(* IEC 61131-3 sources: TA/Tests/RetainTest/At (part 6) *)

(* ---- AtRetainStructureSimple.st ---- *)
PROGRAM AtRetainStructureSimple

AT_RETAINTEST_RETAIN_STRUCTURESIMPLE.AUTO2_BOOL := AT_RETAINTEST_RETAIN_STRUCTURESIMPLE.AUTO1_BOOL;
AT_RETAINTEST_RETAIN_STRUCTURESIMPLE.AUTO2_BYTE := AT_RETAINTEST_RETAIN_STRUCTURESIMPLE.AUTO1_BYTE;
AT_RETAINTEST_RETAIN_STRUCTURESIMPLE.AUTO2_DATE := AT_RETAINTEST_RETAIN_STRUCTURESIMPLE.AUTO1_DATE;
AT_RETAINTEST_RETAIN_STRUCTURESIMPLE.AUTO2_DINT := AT_RETAINTEST_RETAIN_STRUCTURESIMPLE.AUTO1_DINT;
AT_RETAINTEST_RETAIN_STRUCTURESIMPLE.AUTO2_DWORD := AT_RETAINTEST_RETAIN_STRUCTURESIMPLE.AUTO1_DWORD;
AT_RETAINTEST_RETAIN_STRUCTURESIMPLE.AUTO2_INT := AT_RETAINTEST_RETAIN_STRUCTURESIMPLE.AUTO1_INT;
AT_RETAINTEST_RETAIN_STRUCTURESIMPLE.AUTO2_LINT := AT_RETAINTEST_RETAIN_STRUCTURESIMPLE.AUTO1_LINT;
AT_RETAINTEST_RETAIN_STRUCTURESIMPLE.AUTO2_LREAL := AT_RETAINTEST_RETAIN_STRUCTURESIMPLE.AUTO1_LREAL;
AT_RETAINTEST_RETAIN_STRUCTURESIMPLE.AUTO2_LWORD := AT_RETAINTEST_RETAIN_STRUCTURESIMPLE.AUTO1_LWORD;
AT_RETAINTEST_RETAIN_STRUCTURESIMPLE.AUTO2_REAL := AT_RETAINTEST_RETAIN_STRUCTURESIMPLE.AUTO1_REAL;
AT_RETAINTEST_RETAIN_STRUCTURESIMPLE.AUTO2_SINT := AT_RETAINTEST_RETAIN_STRUCTURESIMPLE.AUTO1_SINT;
AT_RETAINTEST_RETAIN_STRUCTURESIMPLE.AUTO2_STRING := AT_RETAINTEST_RETAIN_STRUCTURESIMPLE.AUTO1_STRING;
AT_RETAINTEST_RETAIN_STRUCTURESIMPLE.AUTO2_TIME := AT_RETAINTEST_RETAIN_STRUCTURESIMPLE.AUTO1_TIME;
AT_RETAINTEST_RETAIN_STRUCTURESIMPLE.AUTO2_UDINT := AT_RETAINTEST_RETAIN_STRUCTURESIMPLE.AUTO1_UDINT;
AT_RETAINTEST_RETAIN_STRUCTURESIMPLE.AUTO2_UINT := AT_RETAINTEST_RETAIN_STRUCTURESIMPLE.AUTO1_UINT;
AT_RETAINTEST_RETAIN_STRUCTURESIMPLE.AUTO2_ULINT := AT_RETAINTEST_RETAIN_STRUCTURESIMPLE.AUTO1_ULINT;
AT_RETAINTEST_RETAIN_STRUCTURESIMPLE.AUTO2_USINT := AT_RETAINTEST_RETAIN_STRUCTURESIMPLE.AUTO1_USINT;
AT_RETAINTEST_RETAIN_STRUCTURESIMPLE.AUTO2_WORD := AT_RETAINTEST_RETAIN_STRUCTURESIMPLE.AUTO1_WORD;

AT_RETAINTEST_NONRETAIN_STRUCTURESIMPLE.AUTO2_BOOL := AT_RETAINTEST_NONRETAIN_STRUCTURESIMPLE.AUTO1_BOOL;
AT_RETAINTEST_NONRETAIN_STRUCTURESIMPLE.AUTO2_BYTE := AT_RETAINTEST_NONRETAIN_STRUCTURESIMPLE.AUTO1_BYTE;
AT_RETAINTEST_NONRETAIN_STRUCTURESIMPLE.AUTO2_DATE := AT_RETAINTEST_NONRETAIN_STRUCTURESIMPLE.AUTO1_DATE;
AT_RETAINTEST_NONRETAIN_STRUCTURESIMPLE.AUTO2_DINT := AT_RETAINTEST_NONRETAIN_STRUCTURESIMPLE.AUTO1_DINT;
AT_RETAINTEST_NONRETAIN_STRUCTURESIMPLE.AUTO2_DWORD := AT_RETAINTEST_NONRETAIN_STRUCTURESIMPLE.AUTO1_DWORD;
AT_RETAINTEST_NONRETAIN_STRUCTURESIMPLE.AUTO2_INT := AT_RETAINTEST_NONRETAIN_STRUCTURESIMPLE.AUTO1_INT;
AT_RETAINTEST_NONRETAIN_STRUCTURESIMPLE.AUTO2_LINT := AT_RETAINTEST_NONRETAIN_STRUCTURESIMPLE.AUTO1_LINT;
AT_RETAINTEST_NONRETAIN_STRUCTURESIMPLE.AUTO2_LREAL := AT_RETAINTEST_NONRETAIN_STRUCTURESIMPLE.AUTO1_LREAL;
AT_RETAINTEST_NONRETAIN_STRUCTURESIMPLE.AUTO2_LWORD := AT_RETAINTEST_NONRETAIN_STRUCTURESIMPLE.AUTO1_LWORD;
AT_RETAINTEST_NONRETAIN_STRUCTURESIMPLE.AUTO2_REAL := AT_RETAINTEST_NONRETAIN_STRUCTURESIMPLE.AUTO1_REAL;
AT_RETAINTEST_NONRETAIN_STRUCTURESIMPLE.AUTO2_SINT := AT_RETAINTEST_NONRETAIN_STRUCTURESIMPLE.AUTO1_SINT;
AT_RETAINTEST_NONRETAIN_STRUCTURESIMPLE.AUTO2_STRING := AT_RETAINTEST_NONRETAIN_STRUCTURESIMPLE.AUTO1_STRING;
AT_RETAINTEST_NONRETAIN_STRUCTURESIMPLE.AUTO2_TIME := AT_RETAINTEST_NONRETAIN_STRUCTURESIMPLE.AUTO1_TIME;
AT_RETAINTEST_NONRETAIN_STRUCTURESIMPLE.AUTO2_UDINT := AT_RETAINTEST_NONRETAIN_STRUCTURESIMPLE.AUTO1_UDINT;
AT_RETAINTEST_NONRETAIN_STRUCTURESIMPLE.AUTO2_UINT := AT_RETAINTEST_NONRETAIN_STRUCTURESIMPLE.AUTO1_UINT;
AT_RETAINTEST_NONRETAIN_STRUCTURESIMPLE.AUTO2_ULINT := AT_RETAINTEST_NONRETAIN_STRUCTURESIMPLE.AUTO1_ULINT;
AT_RETAINTEST_NONRETAIN_STRUCTURESIMPLE.AUTO2_USINT := AT_RETAINTEST_NONRETAIN_STRUCTURESIMPLE.AUTO1_USINT;
AT_RETAINTEST_NONRETAIN_STRUCTURESIMPLE.AUTO2_WORD := AT_RETAINTEST_NONRETAIN_STRUCTURESIMPLE.AUTO1_WORD;

AT_RETAINTEST_AUTO_STRUCTURESIMPLE.AUTO2_BOOL := AT_RETAINTEST_AUTO_STRUCTURESIMPLE.AUTO1_BOOL;
AT_RETAINTEST_AUTO_STRUCTURESIMPLE.AUTO2_BYTE := AT_RETAINTEST_AUTO_STRUCTURESIMPLE.AUTO1_BYTE;
AT_RETAINTEST_AUTO_STRUCTURESIMPLE.AUTO2_DATE := AT_RETAINTEST_AUTO_STRUCTURESIMPLE.AUTO1_DATE;
AT_RETAINTEST_AUTO_STRUCTURESIMPLE.AUTO2_DINT := AT_RETAINTEST_AUTO_STRUCTURESIMPLE.AUTO1_DINT;
AT_RETAINTEST_AUTO_STRUCTURESIMPLE.AUTO2_DWORD := AT_RETAINTEST_AUTO_STRUCTURESIMPLE.AUTO1_DWORD;
AT_RETAINTEST_AUTO_STRUCTURESIMPLE.AUTO2_INT := AT_RETAINTEST_AUTO_STRUCTURESIMPLE.AUTO1_INT;
AT_RETAINTEST_AUTO_STRUCTURESIMPLE.AUTO2_LINT := AT_RETAINTEST_AUTO_STRUCTURESIMPLE.AUTO1_LINT;
AT_RETAINTEST_AUTO_STRUCTURESIMPLE.AUTO2_LREAL := AT_RETAINTEST_AUTO_STRUCTURESIMPLE.AUTO1_LREAL;
AT_RETAINTEST_AUTO_STRUCTURESIMPLE.AUTO2_LWORD := AT_RETAINTEST_AUTO_STRUCTURESIMPLE.AUTO1_LWORD;
AT_RETAINTEST_AUTO_STRUCTURESIMPLE.AUTO2_REAL := AT_RETAINTEST_AUTO_STRUCTURESIMPLE.AUTO1_REAL;
AT_RETAINTEST_AUTO_STRUCTURESIMPLE.AUTO2_SINT := AT_RETAINTEST_AUTO_STRUCTURESIMPLE.AUTO1_SINT;
AT_RETAINTEST_AUTO_STRUCTURESIMPLE.AUTO2_STRING := AT_RETAINTEST_AUTO_STRUCTURESIMPLE.AUTO1_STRING;
AT_RETAINTEST_AUTO_STRUCTURESIMPLE.AUTO2_TIME := AT_RETAINTEST_AUTO_STRUCTURESIMPLE.AUTO1_TIME;
AT_RETAINTEST_AUTO_STRUCTURESIMPLE.AUTO2_UDINT := AT_RETAINTEST_AUTO_STRUCTURESIMPLE.AUTO1_UDINT;
AT_RETAINTEST_AUTO_STRUCTURESIMPLE.AUTO2_UINT := AT_RETAINTEST_AUTO_STRUCTURESIMPLE.AUTO1_UINT;
AT_RETAINTEST_AUTO_STRUCTURESIMPLE.AUTO2_ULINT := AT_RETAINTEST_AUTO_STRUCTURESIMPLE.AUTO1_ULINT;
AT_RETAINTEST_AUTO_STRUCTURESIMPLE.AUTO2_USINT := AT_RETAINTEST_AUTO_STRUCTURESIMPLE.AUTO1_USINT;
AT_RETAINTEST_AUTO_STRUCTURESIMPLE.AUTO2_WORD := AT_RETAINTEST_AUTO_STRUCTURESIMPLE.AUTO1_WORD;

END_PROGRAM

(* ---- AtRetainStructureStructureSimple.st ---- *)
PROGRAM AtRetainStructureStructureSimple

AT_RETAINTEST_RETAIN_STRUCTURESTRUCTURESIMPLE.AUTO2.SIMPLE_BOOL := AT_RETAINTEST_RETAIN_STRUCTURESTRUCTURESIMPLE.AUTO1.SIMPLE_BOOL;
AT_RETAINTEST_RETAIN_STRUCTURESTRUCTURESIMPLE.AUTO2.SIMPLE_BYTE := AT_RETAINTEST_RETAIN_STRUCTURESTRUCTURESIMPLE.AUTO1.SIMPLE_BYTE;
AT_RETAINTEST_RETAIN_STRUCTURESTRUCTURESIMPLE.AUTO2.SIMPLE_DATE := AT_RETAINTEST_RETAIN_STRUCTURESTRUCTURESIMPLE.AUTO1.SIMPLE_DATE;
AT_RETAINTEST_RETAIN_STRUCTURESTRUCTURESIMPLE.AUTO2.SIMPLE_DINT := AT_RETAINTEST_RETAIN_STRUCTURESTRUCTURESIMPLE.AUTO1.SIMPLE_DINT;
AT_RETAINTEST_RETAIN_STRUCTURESTRUCTURESIMPLE.AUTO2.SIMPLE_DWORD := AT_RETAINTEST_RETAIN_STRUCTURESTRUCTURESIMPLE.AUTO1.SIMPLE_DWORD;
AT_RETAINTEST_RETAIN_STRUCTURESTRUCTURESIMPLE.AUTO2.SIMPLE_INT := AT_RETAINTEST_RETAIN_STRUCTURESTRUCTURESIMPLE.AUTO1.SIMPLE_INT;
AT_RETAINTEST_RETAIN_STRUCTURESTRUCTURESIMPLE.AUTO2.SIMPLE_LINT := AT_RETAINTEST_RETAIN_STRUCTURESTRUCTURESIMPLE.AUTO1.SIMPLE_LINT;
AT_RETAINTEST_RETAIN_STRUCTURESTRUCTURESIMPLE.AUTO2.SIMPLE_LREAL := AT_RETAINTEST_RETAIN_STRUCTURESTRUCTURESIMPLE.AUTO1.SIMPLE_LREAL;
AT_RETAINTEST_RETAIN_STRUCTURESTRUCTURESIMPLE.AUTO2.SIMPLE_LWORD := AT_RETAINTEST_RETAIN_STRUCTURESTRUCTURESIMPLE.AUTO1.SIMPLE_LWORD;
AT_RETAINTEST_RETAIN_STRUCTURESTRUCTURESIMPLE.AUTO2.SIMPLE_REAL := AT_RETAINTEST_RETAIN_STRUCTURESTRUCTURESIMPLE.AUTO1.SIMPLE_REAL;
AT_RETAINTEST_RETAIN_STRUCTURESTRUCTURESIMPLE.AUTO2.SIMPLE_SINT := AT_RETAINTEST_RETAIN_STRUCTURESTRUCTURESIMPLE.AUTO1.SIMPLE_SINT;
AT_RETAINTEST_RETAIN_STRUCTURESTRUCTURESIMPLE.AUTO2.SIMPLE_STRING := AT_RETAINTEST_RETAIN_STRUCTURESTRUCTURESIMPLE.AUTO1.SIMPLE_STRING;
AT_RETAINTEST_RETAIN_STRUCTURESTRUCTURESIMPLE.AUTO2.SIMPLE_TIME := AT_RETAINTEST_RETAIN_STRUCTURESTRUCTURESIMPLE.AUTO1.SIMPLE_TIME;
AT_RETAINTEST_RETAIN_STRUCTURESTRUCTURESIMPLE.AUTO2.SIMPLE_UDINT := AT_RETAINTEST_RETAIN_STRUCTURESTRUCTURESIMPLE.AUTO1.SIMPLE_UDINT;
AT_RETAINTEST_RETAIN_STRUCTURESTRUCTURESIMPLE.AUTO2.SIMPLE_UINT := AT_RETAINTEST_RETAIN_STRUCTURESTRUCTURESIMPLE.AUTO1.SIMPLE_UINT;
AT_RETAINTEST_RETAIN_STRUCTURESTRUCTURESIMPLE.AUTO2.SIMPLE_ULINT := AT_RETAINTEST_RETAIN_STRUCTURESTRUCTURESIMPLE.AUTO1.SIMPLE_ULINT;
AT_RETAINTEST_RETAIN_STRUCTURESTRUCTURESIMPLE.AUTO2.SIMPLE_USINT := AT_RETAINTEST_RETAIN_STRUCTURESTRUCTURESIMPLE.AUTO1.SIMPLE_USINT;
AT_RETAINTEST_RETAIN_STRUCTURESTRUCTURESIMPLE.AUTO2.SIMPLE_WORD := AT_RETAINTEST_RETAIN_STRUCTURESTRUCTURESIMPLE.AUTO1.SIMPLE_WORD;

AT_RETAINTEST_NONRETAIN_STRUCTURESTRUCTURESIMPLE.AUTO2.SIMPLE_BOOL := AT_RETAINTEST_NONRETAIN_STRUCTURESTRUCTURESIMPLE.AUTO1.SIMPLE_BOOL;
AT_RETAINTEST_NONRETAIN_STRUCTURESTRUCTURESIMPLE.AUTO2.SIMPLE_BYTE := AT_RETAINTEST_NONRETAIN_STRUCTURESTRUCTURESIMPLE.AUTO1.SIMPLE_BYTE;
AT_RETAINTEST_NONRETAIN_STRUCTURESTRUCTURESIMPLE.AUTO2.SIMPLE_DATE := AT_RETAINTEST_NONRETAIN_STRUCTURESTRUCTURESIMPLE.AUTO1.SIMPLE_DATE;
AT_RETAINTEST_NONRETAIN_STRUCTURESTRUCTURESIMPLE.AUTO2.SIMPLE_DINT := AT_RETAINTEST_NONRETAIN_STRUCTURESTRUCTURESIMPLE.AUTO1.SIMPLE_DINT;
AT_RETAINTEST_NONRETAIN_STRUCTURESTRUCTURESIMPLE.AUTO2.SIMPLE_DWORD := AT_RETAINTEST_NONRETAIN_STRUCTURESTRUCTURESIMPLE.AUTO1.SIMPLE_DWORD;
AT_RETAINTEST_NONRETAIN_STRUCTURESTRUCTURESIMPLE.AUTO2.SIMPLE_INT := AT_RETAINTEST_NONRETAIN_STRUCTURESTRUCTURESIMPLE.AUTO1.SIMPLE_INT;
AT_RETAINTEST_NONRETAIN_STRUCTURESTRUCTURESIMPLE.AUTO2.SIMPLE_LINT := AT_RETAINTEST_NONRETAIN_STRUCTURESTRUCTURESIMPLE.AUTO1.SIMPLE_LINT;
AT_RETAINTEST_NONRETAIN_STRUCTURESTRUCTURESIMPLE.AUTO2.SIMPLE_LREAL := AT_RETAINTEST_NONRETAIN_STRUCTURESTRUCTURESIMPLE.AUTO1.SIMPLE_LREAL;
AT_RETAINTEST_NONRETAIN_STRUCTURESTRUCTURESIMPLE.AUTO2.SIMPLE_LWORD := AT_RETAINTEST_NONRETAIN_STRUCTURESTRUCTURESIMPLE.AUTO1.SIMPLE_LWORD;
AT_RETAINTEST_NONRETAIN_STRUCTURESTRUCTURESIMPLE.AUTO2.SIMPLE_REAL := AT_RETAINTEST_NONRETAIN_STRUCTURESTRUCTURESIMPLE.AUTO1.SIMPLE_REAL;
AT_RETAINTEST_NONRETAIN_STRUCTURESTRUCTURESIMPLE.AUTO2.SIMPLE_SINT := AT_RETAINTEST_NONRETAIN_STRUCTURESTRUCTURESIMPLE.AUTO1.SIMPLE_SINT;
AT_RETAINTEST_NONRETAIN_STRUCTURESTRUCTURESIMPLE.AUTO2.SIMPLE_STRING := AT_RETAINTEST_NONRETAIN_STRUCTURESTRUCTURESIMPLE.AUTO1.SIMPLE_STRING;
AT_RETAINTEST_NONRETAIN_STRUCTURESTRUCTURESIMPLE.AUTO2.SIMPLE_TIME := AT_RETAINTEST_NONRETAIN_STRUCTURESTRUCTURESIMPLE.AUTO1.SIMPLE_TIME;
AT_RETAINTEST_NONRETAIN_STRUCTURESTRUCTURESIMPLE.AUTO2.SIMPLE_UDINT := AT_RETAINTEST_NONRETAIN_STRUCTURESTRUCTURESIMPLE.AUTO1.SIMPLE_UDINT;
AT_RETAINTEST_NONRETAIN_STRUCTURESTRUCTURESIMPLE.AUTO2.SIMPLE_UINT := AT_RETAINTEST_NONRETAIN_STRUCTURESTRUCTURESIMPLE.AUTO1.SIMPLE_UINT;
AT_RETAINTEST_NONRETAIN_STRUCTURESTRUCTURESIMPLE.AUTO2.SIMPLE_ULINT := AT_RETAINTEST_NONRETAIN_STRUCTURESTRUCTURESIMPLE.AUTO1.SIMPLE_ULINT;
AT_RETAINTEST_NONRETAIN_STRUCTURESTRUCTURESIMPLE.AUTO2.SIMPLE_USINT := AT_RETAINTEST_NONRETAIN_STRUCTURESTRUCTURESIMPLE.AUTO1.SIMPLE_USINT;
AT_RETAINTEST_NONRETAIN_STRUCTURESTRUCTURESIMPLE.AUTO2.SIMPLE_WORD := AT_RETAINTEST_NONRETAIN_STRUCTURESTRUCTURESIMPLE.AUTO1.SIMPLE_WORD;

AT_RETAINTEST_AUTO_STRUCTURESTRUCTURESIMPLE.AUTO2.SIMPLE_BOOL := AT_RETAINTEST_AUTO_STRUCTURESTRUCTURESIMPLE.AUTO1.SIMPLE_BOOL;
AT_RETAINTEST_AUTO_STRUCTURESTRUCTURESIMPLE.AUTO2.SIMPLE_BYTE := AT_RETAINTEST_AUTO_STRUCTURESTRUCTURESIMPLE.AUTO1.SIMPLE_BYTE;
AT_RETAINTEST_AUTO_STRUCTURESTRUCTURESIMPLE.AUTO2.SIMPLE_DATE := AT_RETAINTEST_AUTO_STRUCTURESTRUCTURESIMPLE.AUTO1.SIMPLE_DATE;
AT_RETAINTEST_AUTO_STRUCTURESTRUCTURESIMPLE.AUTO2.SIMPLE_DINT := AT_RETAINTEST_AUTO_STRUCTURESTRUCTURESIMPLE.AUTO1.SIMPLE_DINT;
AT_RETAINTEST_AUTO_STRUCTURESTRUCTURESIMPLE.AUTO2.SIMPLE_DWORD := AT_RETAINTEST_AUTO_STRUCTURESTRUCTURESIMPLE.AUTO1.SIMPLE_DWORD;
AT_RETAINTEST_AUTO_STRUCTURESTRUCTURESIMPLE.AUTO2.SIMPLE_INT := AT_RETAINTEST_AUTO_STRUCTURESTRUCTURESIMPLE.AUTO1.SIMPLE_INT;
AT_RETAINTEST_AUTO_STRUCTURESTRUCTURESIMPLE.AUTO2.SIMPLE_LINT := AT_RETAINTEST_AUTO_STRUCTURESTRUCTURESIMPLE.AUTO1.SIMPLE_LINT;
AT_RETAINTEST_AUTO_STRUCTURESTRUCTURESIMPLE.AUTO2.SIMPLE_LREAL := AT_RETAINTEST_AUTO_STRUCTURESTRUCTURESIMPLE.AUTO1.SIMPLE_LREAL;
AT_RETAINTEST_AUTO_STRUCTURESTRUCTURESIMPLE.AUTO2.SIMPLE_LWORD := AT_RETAINTEST_AUTO_STRUCTURESTRUCTURESIMPLE.AUTO1.SIMPLE_LWORD;
AT_RETAINTEST_AUTO_STRUCTURESTRUCTURESIMPLE.AUTO2.SIMPLE_REAL := AT_RETAINTEST_AUTO_STRUCTURESTRUCTURESIMPLE.AUTO1.SIMPLE_REAL;
AT_RETAINTEST_AUTO_STRUCTURESTRUCTURESIMPLE.AUTO2.SIMPLE_SINT := AT_RETAINTEST_AUTO_STRUCTURESTRUCTURESIMPLE.AUTO1.SIMPLE_SINT;
AT_RETAINTEST_AUTO_STRUCTURESTRUCTURESIMPLE.AUTO2.SIMPLE_STRING := AT_RETAINTEST_AUTO_STRUCTURESTRUCTURESIMPLE.AUTO1.SIMPLE_STRING;
AT_RETAINTEST_AUTO_STRUCTURESTRUCTURESIMPLE.AUTO2.SIMPLE_TIME := AT_RETAINTEST_AUTO_STRUCTURESTRUCTURESIMPLE.AUTO1.SIMPLE_TIME;
AT_RETAINTEST_AUTO_STRUCTURESTRUCTURESIMPLE.AUTO2.SIMPLE_UDINT := AT_RETAINTEST_AUTO_STRUCTURESTRUCTURESIMPLE.AUTO1.SIMPLE_UDINT;
AT_RETAINTEST_AUTO_STRUCTURESTRUCTURESIMPLE.AUTO2.SIMPLE_UINT := AT_RETAINTEST_AUTO_STRUCTURESTRUCTURESIMPLE.AUTO1.SIMPLE_UINT;
AT_RETAINTEST_AUTO_STRUCTURESTRUCTURESIMPLE.AUTO2.SIMPLE_ULINT := AT_RETAINTEST_AUTO_STRUCTURESTRUCTURESIMPLE.AUTO1.SIMPLE_ULINT;
AT_RETAINTEST_AUTO_STRUCTURESTRUCTURESIMPLE.AUTO2.SIMPLE_USINT := AT_RETAINTEST_AUTO_STRUCTURESTRUCTURESIMPLE.AUTO1.SIMPLE_USINT;
AT_RETAINTEST_AUTO_STRUCTURESTRUCTURESIMPLE.AUTO2.SIMPLE_WORD := AT_RETAINTEST_AUTO_STRUCTURESTRUCTURESIMPLE.AUTO1.SIMPLE_WORD;

END_PROGRAM
